// TIA Portal V17 export
// export: Created 2023-12-22T15:08:06.3852029Z, ExportSetting WithDefaults, DisplayName Totally Integrated Automation Portal, DisplayVersion V17, DisplayName TIA Portal Openness, DisplayVersion V17, DisplayName TIA Portal Version Control Interface, DisplayVersion V17, DisplayName STEP 7 Professional, DisplayVersion V17, DisplayName STEP 7 Safety, DisplayVersion V17, DisplayName WinCC Advanced, DisplayVersion V17
DATA_BLOCK "DIx_1_DB"   // DB200
VERSION : 0.1
// stored: AutoNumber false, DBAccessibleFromOPCUA true, DBAccessibleFromWebserver true, InstanceOfName DIx_1, InstanceOfType FB
"DIx_1"
   // VAR RETAIN
   //    AllBlock { S7_SetPoint := 'True'} : "DI_ex";
   //    FS_Cl_1 { S7_SetPoint := 'True'} : "DI_ex";
   //    FS_Cl_2 { S7_SetPoint := 'True'} : "DI_ex";
   //    PS_PE { S7_SetPoint := 'True'} : "DI_ex";
   //    signal_5 { S7_SetPoint := 'True'} : "DI_ex";
   //    LS_KP_1_1 { S7_SetPoint := 'True'} : "DI_ex";
   //    LS_KP_1_2 { S7_SetPoint := 'True'} : "DI_ex";
   //    LS_KP_2_1 { S7_SetPoint := 'True'} : "DI_ex";
   //    LS_KP_2_2 { S7_SetPoint := 'True'} : "DI_ex";
   //    signal_10 { S7_SetPoint := 'True'} : "DI_ex";
   //    signal_11 { S7_SetPoint := 'True'} : "DI_ex";
   //    signal_12 { S7_SetPoint := 'True'} : "DI_ex";
   //    Time_DTL { S7_SetPoint := 'True'} : DTL := DTL#2023-02-16-09:35:06.552119328;
   // END_VAR
BEGIN
   AllBlock.Use.Inverse := FALSE;
   AllBlock.Use.Indirect := TRUE;
   AllBlock.ADDR_Byte := 0;
   AllBlock.ADDR_Bit := 9;
   AllBlock.Filter_On.SP := 16#02;
   AllBlock.Filter_Off.SP := 16#02;
   FS_Cl_1.Use.Inverse := TRUE;
   FS_Cl_1.Use.Indirect := TRUE;
   FS_Cl_1.ADDR_Byte := 3;
   FS_Cl_1.ADDR_Bit := 6;
   FS_Cl_1.Filter_On.SP := 16#02;
   FS_Cl_1.Filter_Off.SP := 16#02;
   FS_Cl_2.Use.Inverse := TRUE;
   FS_Cl_2.Use.Indirect := TRUE;
   FS_Cl_2.ADDR_Byte := 3;
   FS_Cl_2.ADDR_Bit := 7;
   FS_Cl_2.Filter_On.SP := 16#02;
   FS_Cl_2.Filter_Off.SP := 16#02;
   PS_PE.Use.Inverse := FALSE;
   PS_PE.Use.Indirect := TRUE;
   PS_PE.ADDR_Byte := 0;
   PS_PE.ADDR_Bit := 9;
   PS_PE.Filter_On.SP := 16#02;
   PS_PE.Filter_Off.SP := 16#02;
   signal_5.Use.Inverse := FALSE;
   signal_5.Use.Indirect := TRUE;
   signal_5.ADDR_Byte := 0;
   signal_5.ADDR_Bit := 9;
   signal_5.Filter_On.SP := 16#02;
   signal_5.Filter_Off.SP := 16#02;
   LS_KP_1_1.Use.Inverse := FALSE;
   LS_KP_1_1.Use.Indirect := TRUE;
   LS_KP_1_1.ADDR_Byte := 4;
   LS_KP_1_1.ADDR_Bit := 2;
   LS_KP_1_1.Filter_On.SP := 16#02;
   LS_KP_1_1.Filter_Off.SP := 16#02;
   LS_KP_1_2.Use.Inverse := FALSE;
   LS_KP_1_2.Use.Indirect := TRUE;
   LS_KP_1_2.ADDR_Byte := 4;
   LS_KP_1_2.ADDR_Bit := 3;
   LS_KP_1_2.Filter_On.SP := 16#02;
   LS_KP_1_2.Filter_Off.SP := 16#02;
   LS_KP_2_1.Use.Inverse := FALSE;
   LS_KP_2_1.Use.Indirect := TRUE;
   LS_KP_2_1.ADDR_Byte := 4;
   LS_KP_2_1.ADDR_Bit := 4;
   LS_KP_2_1.Filter_On.SP := 16#02;
   LS_KP_2_1.Filter_Off.SP := 16#02;
   LS_KP_2_2.Use.Inverse := FALSE;
   LS_KP_2_2.Use.Indirect := TRUE;
   LS_KP_2_2.ADDR_Byte := 4;
   LS_KP_2_2.ADDR_Bit := 5;
   LS_KP_2_2.Filter_On.SP := 16#02;
   LS_KP_2_2.Filter_Off.SP := 16#02;
   signal_10.Use.Inverse := FALSE;
   signal_10.Use.Indirect := TRUE;
   signal_10.ADDR_Byte := 0;
   signal_10.ADDR_Bit := 9;
   signal_10.Filter_On.SP := 16#02;
   signal_10.Filter_Off.SP := 16#02;
   signal_11.Use.Inverse := FALSE;
   signal_11.Use.Indirect := TRUE;
   signal_11.ADDR_Byte := 0;
   signal_11.ADDR_Bit := 9;
   signal_11.Filter_On.SP := 16#02;
   signal_11.Filter_Off.SP := 16#02;
   signal_12.Use.Inverse := FALSE;
   signal_12.Use.Indirect := TRUE;
   signal_12.ADDR_Byte := 0;
   signal_12.ADDR_Bit := 9;
   signal_12.Filter_On.SP := 16#02;
   signal_12.Filter_Off.SP := 16#02;
END_DATA_BLOCK
